FUNCTION_BLOCK FB_Conveyor
VAR_INPUT
	bEnable : BOOL;
END_VAR
VAR_OUTPUT
	bFull : BOOL;
	bMoving : BOOL;
END_VAR
VAR
	fbAxis : FB_Axis;
	iCount : INT;
END_VAR

fbAxis(bEnable := bEnable, fVelocity := 120.0, fAcceleration := 400.0);
bMoving := fbAxis.bBusy;
bFull := iCount > 20;
iCount := iCount + 1;

METHOD PUBLIC Reset : BOOL
VAR
	i : INT;
END_VAR
iCount := 0;
bFull := FALSE;
Reset := TRUE;
END_METHOD

METHOD PUBLIC SetSpeed : BOOL
VAR_INPUT
	fSpeed : LREAL;
END_VAR
// A speed above the mechanical limit is rejected rather
// than passed on, so the axis never sees an unreachable target.
IF fSpeed > 0.0 AND fSpeed <= 2000.0 THEN
	fbAxis(bEnable := TRUE, fVelocity := fSpeed, fAcceleration := 400.0);
	SetSpeed := TRUE;
ELSE
	SetSpeed := FALSE;
END_IF
END_METHOD

PROPERTY PUBLIC Count : INT
GET
GET
END_GET
SET
SET
END_SET
END_PROPERTY

END_FUNCTION_BLOCK

FUNCTION_BLOCK FB_Picker
VAR_INPUT
	bEnable : BOOL;
	iCode : UINT;
END_VAR
VAR_OUTPUT
	bDone : BOOL;
END_VAR

bDone := NOT bEnable;
IF bEnable AND iCode = 16#0 THEN
	bDone := TRUE;
END_IF

END_FUNCTION_BLOCK

(* stored: Version 1.1.0.1
   POU FB_Conveyor: Id {7a3f2c10-4b8e-4c1a-9f20-1d5e6b7a8c90}, SpecialFunc None
   Method Reset: Id {1b2c3d4e-5f60-4718-8293-a4b5c6d7e8f9}
   Method SetSpeed: Id {2c3d4e5f-6071-4829-93a4-b5c6d7e8f901}
   Property Count: Id {3d4e5f60-7182-493a-b4c5-d6e7f8091a2b}
   POU FB_Picker: Id {4e5f6071-8293-4a4b-95c6-d7e8f9012a3b}, SpecialFunc None *)
